PROGRAM posCarrinho3
VAR
	timeCalc: TIME;
	bNotificaTime: BOOL:= TRUE;
END_VAR


///// CALCULO DE DEFINIÇÃO SE O PROCESSO PASSA DAS 36 HORAS LIMITES ----------------------------------------
timeCalc:= (gvl_p.arrStatusEstufas[2].prevFimSeca - systemtime_to_dt(gvl.fbGetLocalSystemTime.systemTime));
IF timeCalc < T#24H and bNotificaTime THEN
	bNotificaTime:= FALSE;
	ELSE
		bNotificaTime:= TRUE;
		
END_IF

END_PROGRAM

(* stored: Version 1.1.0.1, ProductVersion 3.1.4024.12
   POU posCarrinho3: Id {edddb965-295a-4cb5-996b-c47f3d2fc46f}, SpecialFunc None *)
